// TwinCAT 3 PLC project PLC1
// ProgramVersion: 3.1.4022.0
// libraries:
//   Tc2_Standard, * (Beckhoff Automation GmbH)
//   Tc2_System, * (Beckhoff Automation GmbH)
//   Tc3_Module, * (Beckhoff Automation GmbH)
// project tree:
//   DUTs/ DUT.TcDUT, HOIST_REF_OpcToPlc.TcDUT, HOIST_REF_PlcToOpc.TcDUT
//   GVLs/ Grinder.TcGVL, GVL_HOIST.TcGVL
//   / PlcTask.TcTTO
//   POUs/ MAIN.TcPOU
// real-time tasks:
//   TASK PlcTask: cycle T#1ms, priority 20, ADS port 350

CONFIGURATION PLC1
    RESOURCE PLC ON TwinCAT3
        TASK PlcTask(INTERVAL := T#1ms, PRIORITY := 20);
        PROGRAM MAIN WITH PlcTask : MAIN;
    END_RESOURCE
END_CONFIGURATION

// ---- DUTs/DUT.TcDUT
TYPE DUT :
STRUCT
	aStartPoint  : INT;
    aPoint1      : INT;
    aPoint2      : INT;
    aPoint3      : INT;
    aPoint4      : INT;
    aEndPoint    : INT;
END_STRUCT
END_TYPE

// ---- DUTs/HOIST_REF_OpcToPlc.TcDUT
TYPE HOIST_REF_OpcToPlc :
STRUCT
	DestPos	:	REAL;
	DestVel	:	REAL;
END_STRUCT
END_TYPE

// ---- DUTs/HOIST_REF_PlcToOpc.TcDUT

TYPE HOIST_REF_PlcToOpc :
STRUCT
	ActPos	:	REAL;
	ActVel	:	REAL;
	EndPosUp	: BOOL;
	EndPosDown	: BOOL;
	
END_STRUCT
END_TYPE

// ---- GVLs/Grinder.TcGVL
{attribute 'qualified_only'}
VAR_GLOBAL
	GrindingWheelMS:BOOL;
	GrindingWheelMS2:BOOL;
END_VAR

// ---- GVLs/GVL_HOIST.TcGVL

VAR_GLOBAL
	{attribute 'OPC.UA.DA' := '1'} 
	stHoistOpcToPlc				: ARRAY[1..cHoistCount] OF HOIST_REF_OpcToPlc;
	{attribute 'OPC.UA.DA' := '1'} 
	stHoistPlcToOpc				: ARRAY[1..cHoistCount] OF HOIST_REF_PlcToOpc;
END_VAR
VAR_GLOBAL CONSTANT
	cHoistCount			: UINT:=255;
END_VAR

// ---- POUs/MAIN.TcPOU
PROGRAM MAIN
VAR
	{attribute 'OPC.UA.DA' := '1'} 
	increment:INT;
	GrindingWheelMS: BOOL;
	{attribute 'OPC.UA.DA' := '1'} 
	GrindingWheelMS2: BOOL;
	{attribute 'OPC.UA.DA' := '1'} 
	ex_struct: DUT;
	{attribute 'OPC.UA.DA' := '1'}
	arr1 : ARRAY [1..256] OF INT;
	{attribute 'OPC.UA.DA' := '1'}
	count: INT;
	counter: INT;
END_VAR

increment:=increment+1;
GrindingWheelMS:=TRUE;
GrindingWheelMS2:=FALSE;
ex_struct.aPoint1:=2;
ex_struct.aPoint2:=5;
ex_struct.aPoint3:=6;
ex_struct.aPoint4:=12;
ex_struct.aEndPoint:=24;
ex_struct.aStartPoint:=1;

counter := counter + 1;
arr1[counter] := counter + increment;
stHoistPlcToOpc[counter].ActPos := increment;
IF counter > 254 THEN
	counter := 0;
END_IF;

END_PROGRAM
